// TIA Portal V17 export
// export: Created 2022-03-12T16:05:15.4162152Z, ExportSetting WithDefaults, DisplayName Totally Integrated Automation Portal, DisplayVersion V17, DisplayName TIA Portal Openness, DisplayVersion V17, DisplayName TIA Portal Version Control Interface, DisplayVersion V17, DisplayName STEP 7 Professional, DisplayVersion V17, DisplayName STEP 7 Safety, DisplayVersion V17, DisplayName WinCC Advanced / Unified PC, DisplayVersion V17
FUNCTION_BLOCK "UN_05_EventSummation"   // FB31625, LAD
TITLE = UN_05_EventSummation
{ S7_Optimized_Access := 'TRUE' }
AUTHOR : tech.team.motioncontrol@siemens.com
FAMILY : CPG
VERSION : 1.1
// Support: tech.team.motioncontrol@siemens.com
// stored: AutoNumber true, IsIECCheckEnabled false, IsRetainMemResEnabled false, MemoryReserve 100, SetENOAutomatically false, UDAEnableTagReadback false
   VAR
      instEventSumBeg_Alarm { S7_SetPoint := 'True'} : "CPG_EventSummationBegin";   // instanceFB - EventSummationBegin - Alarm Events
      instEventSum_Alarm_UN { S7_SetPoint := 'True'} : "CPG_EventSummation";   // instanceFB - EventSummation FB - Alarm Events - UN
      instEventSum_Alarm_EM00 { S7_SetPoint := 'True'} : "CPG_EventSummation";   // instanceFB - EventSummation FB - Alarm Events - EM00
      instEventSum_Alarm_EM01 { S7_SetPoint := 'True'} : "CPG_EventSummation";   // instanceFB - EventSummation FB - Alarm Events - EM01
      instEventSum_Alarm_EM02 { S7_SetPoint := 'True'} : "CPG_EventSummation";   // instanceFB - EventSummation FB - Alarm Events - EM02
      instEventSumEnd_Alarm { S7_SetPoint := 'True'} : "CPG_EventSummationEnd";   // instanceFB - EventSummationEnd - Alarm Events
      instEventSortFilter_Alarm { S7_SetPoint := 'True'} : "CPG_EventSortFilter";   // instanceFB - EventSortFilter FB - Alarms
      instAlarmMove { S7_SetPoint := 'True'} : "CPG_AlarmMove";   // instance FB - Alarm Move
      instEventSumBeg_Warning { S7_SetPoint := 'True'} : "CPG_EventSummationBegin";   // instanceFB - EventSummationBegin - Warning Events
      instEventSum_Warning_UN { S7_SetPoint := 'True'} : "CPG_EventSummation";   // instanceFB - EventSummation FB - Warning Events - UN
      instEventSum_Warning_EM00 { S7_SetPoint := 'True'} : "CPG_EventSummation";   // instanceFB - EventSummation FB - Warning Events - EM00
      instEventSum_Warning_EM01 { S7_SetPoint := 'True'} : "CPG_EventSummation";   // instanceFB - EventSummation FB - Warning Events - EM01
      instEventSum_Warning_EM02 { S7_SetPoint := 'True'} : "CPG_EventSummation";   // instanceFB - EventSummation FB - Warning Events - EM02
      instEventSumEnd_Warning { S7_SetPoint := 'True'} : "CPG_EventSummationEnd";   // instanceFB - EventSummationEnd - Warning Events
      instEventSortFilter_Warning { S7_SetPoint := 'True'} : "CPG_EventSortFilter";   // instanceFB - EventSortFilter FB - Alarms
      instWarning_MsgScroll { S7_SetPoint := 'True'} : "CPG_MsgScroll";   // instance FB - Warning Scroll
      instEventSumBeg_Status { S7_SetPoint := 'True'} : "CPG_EventSummationBegin";   // instanceFB - EventSummationBegin - Status Events
      instEventSum_Status_UN { S7_SetPoint := 'True'} : "CPG_EventSummation";   // instanceFB - EventSummation FB - Status Events - UN
      instEventSum_Status_EM00 { S7_SetPoint := 'True'} : "CPG_EventSummation";   // instanceFB - EventSummation FB - Status Events - EM00
      instEventSum_Status_EM01 { S7_SetPoint := 'True'} : "CPG_EventSummation";   // instanceFB - EventSummation FB - Status Events - EM01
      instEventSum_Status_EM02 { S7_SetPoint := 'True'} : "CPG_EventSummation";   // instanceFB - EventSummation FB - Status Events - EM02
      instEventSumEnd_Status { S7_SetPoint := 'True'} : "CPG_EventSummationEnd";   // instanceFB - EventSummationEnd - Status Events
      instPackML_AlarmHistory { S7_SetPoint := 'True'} : "CPG_AlarmHistory";   // instance FB - Capturing the 1st fault history
      instProgram_Alarm { S7_SetPoint := 'True'} : Program_Alarm;   // instance DB for Program Alarm - diag to PLC HMI
      instWarningMove { S7_SetPoint := 'True'} : "CPG_AlarmMove";
      instPareto { S7_SetPoint := 'True'} : "CPG_ParetoAnalysis";
   END_VAR
   VAR_TEMP
      tempAlarmMove_Sts_Error : Bool;   // Error with AlarmMove?
      tempAlarmMove_Sts_ErrorCode : Int;   // AlarmMove Error code
      tempProgramAlarm_error : Bool;
      tempProgramAlarm_status : Word;
   END_VAR
BEGIN

REGION Network 1: Call the Alarm Event Summary - Beginning FB
   // **********  ALARM CONTROL SUMMATION  **********
   //  
   // The event summation begin instruction prepares the summation blocks.  It should 
   // be run each time before the FB_EventSummation blocks.
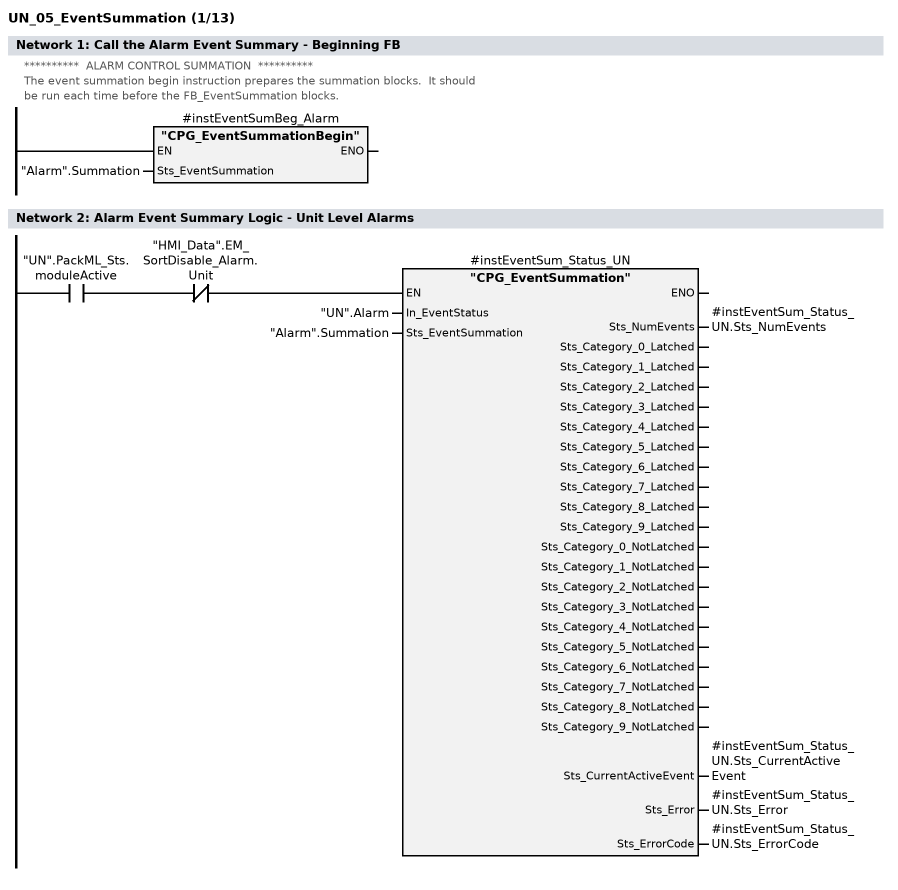
   RUNG wire#powerrail
      #instEventSumBeg_Alarm(Sts_EventSummation := "Alarm".Summation)
   END_RUNG
   // the same network as SCL:
   #instEventSumBeg_Alarm(Sts_EventSummation := "Alarm".Summation);   // "CPG_EventSummationBegin"
END_REGION

REGION Network 2: Alarm Event Summary Logic - Unit Level Alarms
   RUNG wire#powerrail
      Contact( "UN".PackML_Sts.moduleActive )
      I_Contact( "HMI_Data".EM_SortDisable_Alarm.Unit )
      #instEventSum_Status_UN(In_EventStatus := "UN".Alarm, Sts_EventSummation := "Alarm".Summation, Sts_NumEvents => #instEventSum_Status_UN.Sts_NumEvents, Sts_Category_0_Latched =>, Sts_Category_1_Latched =>, Sts_Category_2_Latched =>, Sts_Category_3_Latched =>, Sts_Category_4_Latched =>, Sts_Category_5_Latched =>, Sts_Category_6_Latched =>, Sts_Category_7_Latched =>, Sts_Category_8_Latched =>, Sts_Category_9_Latched =>, Sts_Category_0_NotLatched =>, Sts_Category_1_NotLatched =>, Sts_Category_2_NotLatched =>, Sts_Category_3_NotLatched =>, Sts_Category_4_NotLatched =>, Sts_Category_5_NotLatched =>, Sts_Category_6_NotLatched =>, Sts_Category_7_NotLatched =>, Sts_Category_8_NotLatched =>, Sts_Category_9_NotLatched =>, Sts_CurrentActiveEvent => #instEventSum_Status_UN.Sts_CurrentActiveEvent, Sts_Error => #instEventSum_Status_UN.Sts_Error, Sts_ErrorCode => #instEventSum_Status_UN.Sts_ErrorCode)
   END_RUNG
   // the same network as SCL:
   IF "UN".PackML_Sts.moduleActive AND NOT "HMI_Data".EM_SortDisable_Alarm.Unit THEN
       #instEventSum_Status_UN(In_EventStatus := "UN".Alarm,   // "CPG_EventSummation"
                               Sts_EventSummation := "Alarm".Summation,
                               Sts_NumEvents => #instEventSum_Status_UN.Sts_NumEvents,
                               Sts_CurrentActiveEvent => #instEventSum_Status_UN.Sts_CurrentActiveEvent,
                               Sts_Error => #instEventSum_Status_UN.Sts_Error,
                               Sts_ErrorCode => #instEventSum_Status_UN.Sts_ErrorCode);
   END_IF;
END_REGION

REGION Network 3: Alarm Event Summary Logic - Equipment Module #00
   // This instance of the Event Sum (or Event Summation) is used to merge the events 
   // from EM0 into the larger Unit or UN evevts list.
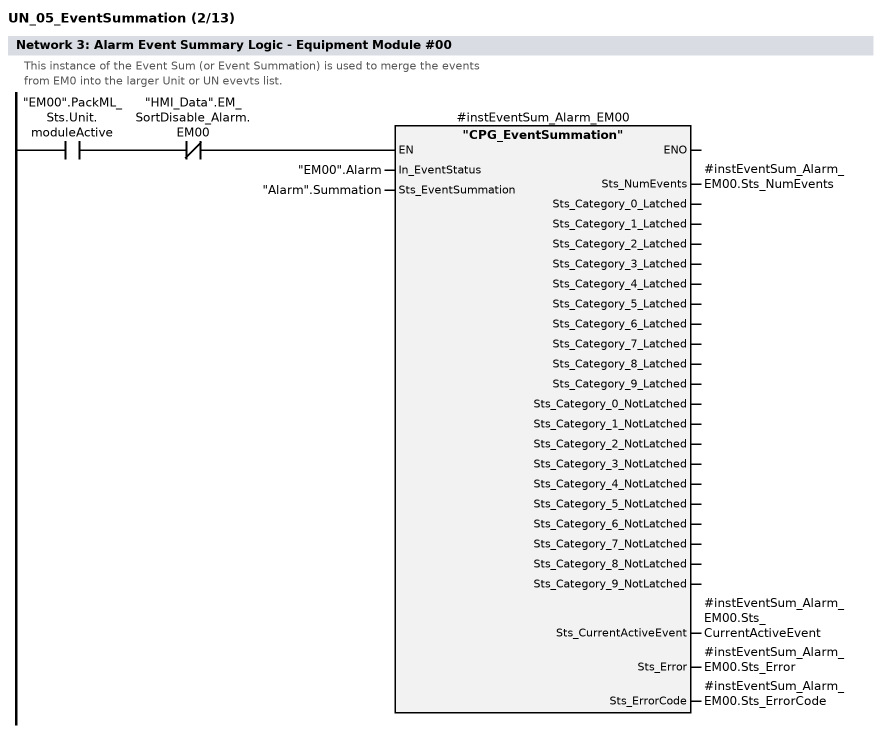
   RUNG wire#powerrail
      Contact( "EM00".PackML_Sts.Unit.moduleActive )
      I_Contact( "HMI_Data".EM_SortDisable_Alarm.EM00 )
      #instEventSum_Alarm_EM00(In_EventStatus := "EM00".Alarm, Sts_EventSummation := "Alarm".Summation, Sts_NumEvents => #instEventSum_Alarm_EM00.Sts_NumEvents, Sts_Category_0_Latched =>, Sts_Category_1_Latched =>, Sts_Category_2_Latched =>, Sts_Category_3_Latched =>, Sts_Category_4_Latched =>, Sts_Category_5_Latched =>, Sts_Category_6_Latched =>, Sts_Category_7_Latched =>, Sts_Category_8_Latched =>, Sts_Category_9_Latched =>, Sts_Category_0_NotLatched =>, Sts_Category_1_NotLatched =>, Sts_Category_2_NotLatched =>, Sts_Category_3_NotLatched =>, Sts_Category_4_NotLatched =>, Sts_Category_5_NotLatched =>, Sts_Category_6_NotLatched =>, Sts_Category_7_NotLatched =>, Sts_Category_8_NotLatched =>, Sts_Category_9_NotLatched =>, Sts_CurrentActiveEvent => #instEventSum_Alarm_EM00.Sts_CurrentActiveEvent, Sts_Error => #instEventSum_Alarm_EM00.Sts_Error, Sts_ErrorCode => #instEventSum_Alarm_EM00.Sts_ErrorCode)
   END_RUNG
   // the same network as SCL:
   IF "EM00".PackML_Sts.Unit.moduleActive AND NOT "HMI_Data".EM_SortDisable_Alarm.EM00 THEN
       #instEventSum_Alarm_EM00(In_EventStatus := "EM00".Alarm,   // "CPG_EventSummation"
                               Sts_EventSummation := "Alarm".Summation,
                               Sts_NumEvents => #instEventSum_Alarm_EM00.Sts_NumEvents,
                               Sts_CurrentActiveEvent => #instEventSum_Alarm_EM00.Sts_CurrentActiveEvent,
                               Sts_Error => #instEventSum_Alarm_EM00.Sts_Error,
                               Sts_ErrorCode => #instEventSum_Alarm_EM00.Sts_ErrorCode);
   END_IF;
END_REGION

REGION Network 4: Alarm Event Summary Logic - Equipment Module #01
   // This instance of the Event Sum (or Event Summation) is used to merge the events 
   // from EM01 into the larger Unit or UN evevts list.
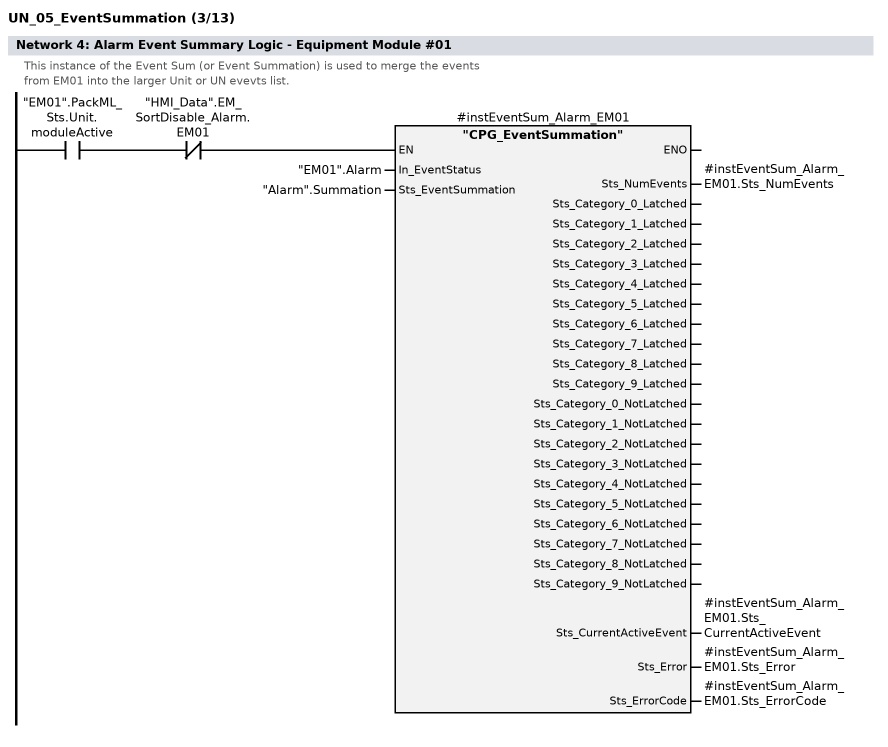
   RUNG wire#powerrail
      Contact( "EM01".PackML_Sts.Unit.moduleActive )
      I_Contact( "HMI_Data".EM_SortDisable_Alarm.EM01 )
      #instEventSum_Alarm_EM01(In_EventStatus := "EM01".Alarm, Sts_EventSummation := "Alarm".Summation, Sts_NumEvents => #instEventSum_Alarm_EM01.Sts_NumEvents, Sts_Category_0_Latched =>, Sts_Category_1_Latched =>, Sts_Category_2_Latched =>, Sts_Category_3_Latched =>, Sts_Category_4_Latched =>, Sts_Category_5_Latched =>, Sts_Category_6_Latched =>, Sts_Category_7_Latched =>, Sts_Category_8_Latched =>, Sts_Category_9_Latched =>, Sts_Category_0_NotLatched =>, Sts_Category_1_NotLatched =>, Sts_Category_2_NotLatched =>, Sts_Category_3_NotLatched =>, Sts_Category_4_NotLatched =>, Sts_Category_5_NotLatched =>, Sts_Category_6_NotLatched =>, Sts_Category_7_NotLatched =>, Sts_Category_8_NotLatched =>, Sts_Category_9_NotLatched =>, Sts_CurrentActiveEvent => #instEventSum_Alarm_EM01.Sts_CurrentActiveEvent, Sts_Error => #instEventSum_Alarm_EM01.Sts_Error, Sts_ErrorCode => #instEventSum_Alarm_EM01.Sts_ErrorCode)
   END_RUNG
   // the same network as SCL:
   IF "EM01".PackML_Sts.Unit.moduleActive AND NOT "HMI_Data".EM_SortDisable_Alarm.EM01 THEN
       #instEventSum_Alarm_EM01(In_EventStatus := "EM01".Alarm,   // "CPG_EventSummation"
                               Sts_EventSummation := "Alarm".Summation,
                               Sts_NumEvents => #instEventSum_Alarm_EM01.Sts_NumEvents,
                               Sts_CurrentActiveEvent => #instEventSum_Alarm_EM01.Sts_CurrentActiveEvent,
                               Sts_Error => #instEventSum_Alarm_EM01.Sts_Error,
                               Sts_ErrorCode => #instEventSum_Alarm_EM01.Sts_ErrorCode);
   END_IF;
END_REGION

REGION Network 5: Alarm Event Summary Logic - Equipment Module #02
   // This instance of the Event Sum (or Event Summation) is used to merge the events 
   // from EM01 into the larger Unit or UN evevts list.
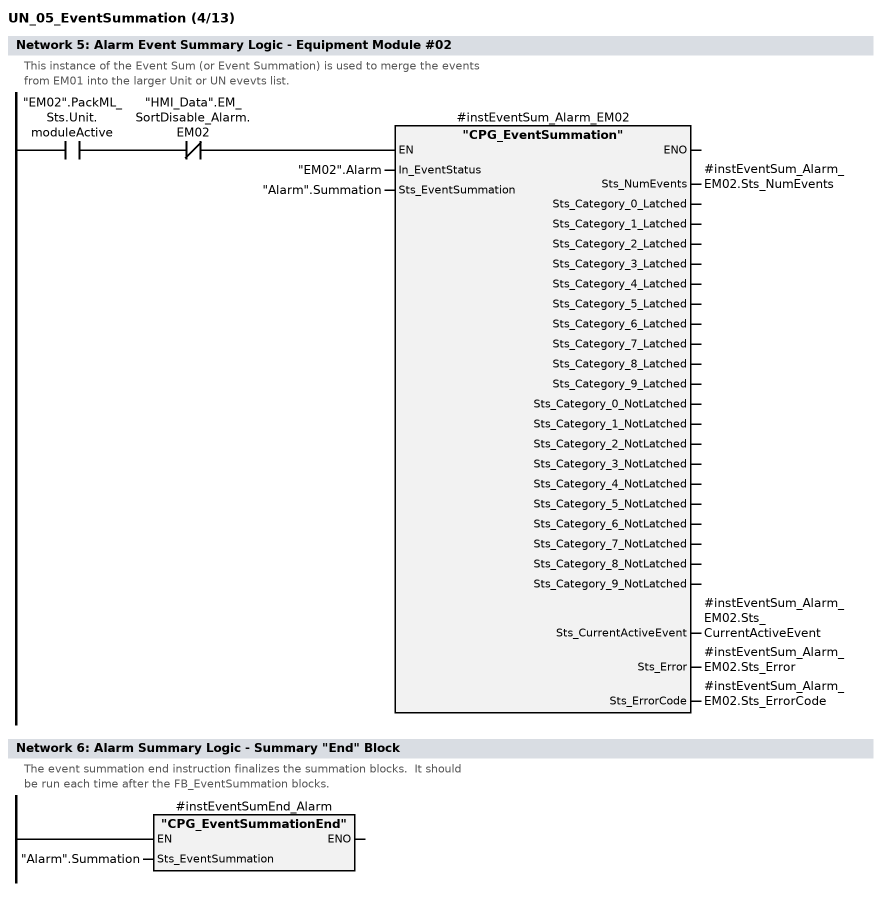
   RUNG wire#powerrail
      Contact( "EM02".PackML_Sts.Unit.moduleActive )
      I_Contact( "HMI_Data".EM_SortDisable_Alarm.EM02 )
      #instEventSum_Alarm_EM02(In_EventStatus := "EM02".Alarm, Sts_EventSummation := "Alarm".Summation, Sts_NumEvents => #instEventSum_Alarm_EM02.Sts_NumEvents, Sts_Category_0_Latched =>, Sts_Category_1_Latched =>, Sts_Category_2_Latched =>, Sts_Category_3_Latched =>, Sts_Category_4_Latched =>, Sts_Category_5_Latched =>, Sts_Category_6_Latched =>, Sts_Category_7_Latched =>, Sts_Category_8_Latched =>, Sts_Category_9_Latched =>, Sts_Category_0_NotLatched =>, Sts_Category_1_NotLatched =>, Sts_Category_2_NotLatched =>, Sts_Category_3_NotLatched =>, Sts_Category_4_NotLatched =>, Sts_Category_5_NotLatched =>, Sts_Category_6_NotLatched =>, Sts_Category_7_NotLatched =>, Sts_Category_8_NotLatched =>, Sts_Category_9_NotLatched =>, Sts_CurrentActiveEvent => #instEventSum_Alarm_EM02.Sts_CurrentActiveEvent, Sts_Error => #instEventSum_Alarm_EM02.Sts_Error, Sts_ErrorCode => #instEventSum_Alarm_EM02.Sts_ErrorCode)
   END_RUNG
   // the same network as SCL:
   IF "EM02".PackML_Sts.Unit.moduleActive AND NOT "HMI_Data".EM_SortDisable_Alarm.EM02 THEN
       #instEventSum_Alarm_EM02(In_EventStatus := "EM02".Alarm,   // "CPG_EventSummation"
                               Sts_EventSummation := "Alarm".Summation,
                               Sts_NumEvents => #instEventSum_Alarm_EM02.Sts_NumEvents,
                               Sts_CurrentActiveEvent => #instEventSum_Alarm_EM02.Sts_CurrentActiveEvent,
                               Sts_Error => #instEventSum_Alarm_EM02.Sts_Error,
                               Sts_ErrorCode => #instEventSum_Alarm_EM02.Sts_ErrorCode);
   END_IF;
END_REGION

REGION Network 6: Alarm Summary Logic - Summary "End" Block
   // The event summation end instruction finalizes the summation blocks.  It should 
   // be run each time after the FB_EventSummation blocks.
   RUNG wire#powerrail
      #instEventSumEnd_Alarm(Sts_EventSummation := "Alarm".Summation)
   END_RUNG
   // the same network as SCL:
   #instEventSumEnd_Alarm(Sts_EventSummation := "Alarm".Summation);   // "CPG_EventSummationEnd"
END_REGION

REGION Network 7: Update Admin.Alarm information.
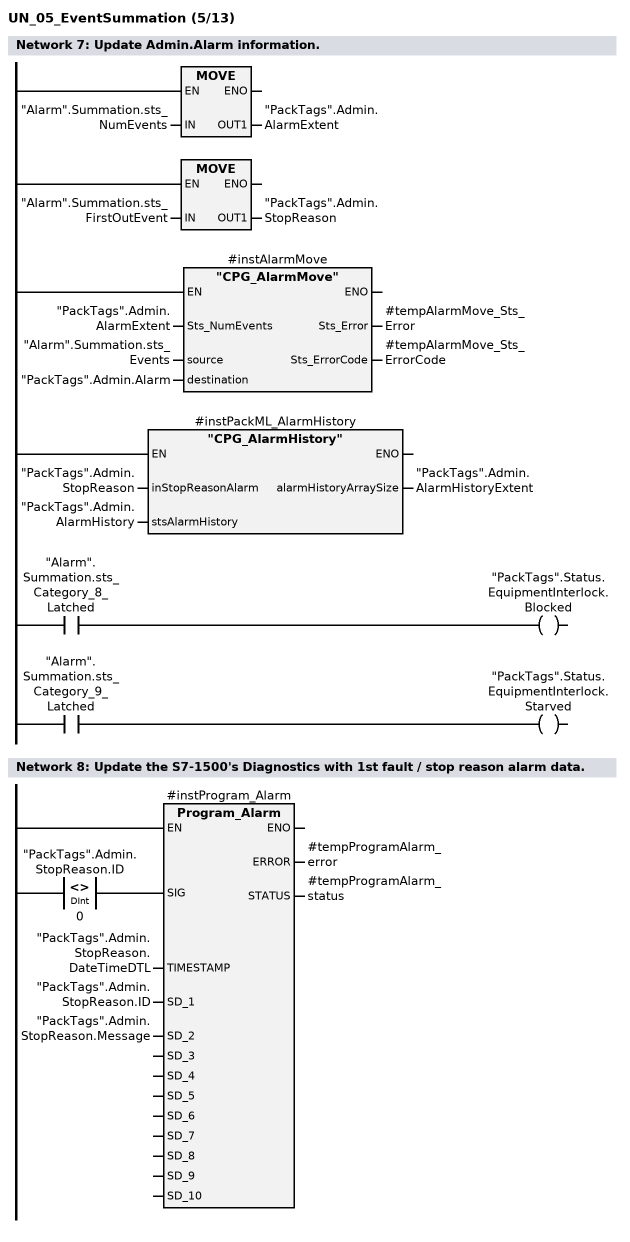
   RUNG wire#powerrail
      { S7_GenerateENO := "TRUE" } Move(in := "Alarm".Summation.sts_NumEvents, out1 => "PackTags".Admin.AlarmExtent)
   END_RUNG
   RUNG wire#powerrail
      Move(in := "Alarm".Summation.sts_FirstOutEvent, out1 => "PackTags".Admin.StopReason)
   END_RUNG
   RUNG wire#powerrail
      #instAlarmMove(Sts_NumEvents := "PackTags".Admin.AlarmExtent, source := "Alarm".Summation.sts_Events, destination := "PackTags".Admin.Alarm, Sts_Error => #tempAlarmMove_Sts_Error, Sts_ErrorCode => #tempAlarmMove_Sts_ErrorCode)
   END_RUNG
   RUNG wire#powerrail
      #instPackML_AlarmHistory(inStopReasonAlarm := "PackTags".Admin.StopReason, stsAlarmHistory := "PackTags".Admin.AlarmHistory, alarmHistoryArraySize => "PackTags".Admin.AlarmHistoryExtent)
   END_RUNG
   RUNG wire#powerrail
      Contact( "Alarm".Summation.sts_Category_8_Latched )
      Coil( "PackTags".Status.EquipmentInterlock.Blocked )
   END_RUNG
   RUNG wire#powerrail
      Contact( "Alarm".Summation.sts_Category_9_Latched )
      Coil( "PackTags".Status.EquipmentInterlock.Starved )
   END_RUNG
   // the same network as SCL:
   "PackTags".Admin.AlarmExtent := "Alarm".Summation.sts_NumEvents;
   "PackTags".Admin.StopReason := "Alarm".Summation.sts_FirstOutEvent;
   #instAlarmMove(Sts_NumEvents := "PackTags".Admin.AlarmExtent,   // "CPG_AlarmMove"
                  source := "Alarm".Summation.sts_Events,
                  destination := "PackTags".Admin.Alarm,
                  Sts_Error => #tempAlarmMove_Sts_Error,
                  Sts_ErrorCode => #tempAlarmMove_Sts_ErrorCode);
   #instPackML_AlarmHistory(inStopReasonAlarm := "PackTags".Admin.StopReason,   // "CPG_AlarmHistory"
                           stsAlarmHistory := "PackTags".Admin.AlarmHistory,
                           alarmHistoryArraySize => "PackTags".Admin.AlarmHistoryExtent);
   "PackTags".Status.EquipmentInterlock.Blocked := "Alarm".Summation.sts_Category_8_Latched;
   "PackTags".Status.EquipmentInterlock.Starved := "Alarm".Summation.sts_Category_9_Latched;
END_REGION

REGION Network 8: Update the S7-1500's Diagnostics with 1st fault / stop reason alarm data.
   RUNG wire#powerrail
      #instProgram_Alarm.Program_Alarm(SIG := wire#w1, TIMESTAMP := "PackTags".Admin.StopReason.DateTimeDTL, SD_1 := "PackTags".Admin.StopReason.ID, SD_2 := "PackTags".Admin.StopReason.Message, SD_3 :=, SD_4 :=, SD_5 :=, SD_6 :=, SD_7 :=, SD_8 :=, SD_9 :=, SD_10 :=, Error => #tempProgramAlarm_error, Status => #tempProgramAlarm_status)
   END_RUNG
   RUNG wire#powerrail
      { S7_Templates := "SrcType := DInt" } NE_Contact(in1 := "PackTags".Admin.StopReason.ID, in2 := 0)
   END_RUNG wire#w1
   // the same network as SCL:
   #instProgram_Alarm(SIG := "PackTags".Admin.StopReason.ID <> 0,   // Program_Alarm
                      TIMESTAMP := "PackTags".Admin.StopReason.DateTimeDTL,
                      SD_1 := "PackTags".Admin.StopReason.ID,
                      SD_2 := "PackTags".Admin.StopReason.Message,
                      Error => #tempProgramAlarm_error,
                      Status => #tempProgramAlarm_status);
END_REGION

REGION Network 9: Event Sort Filter logic - Alarms
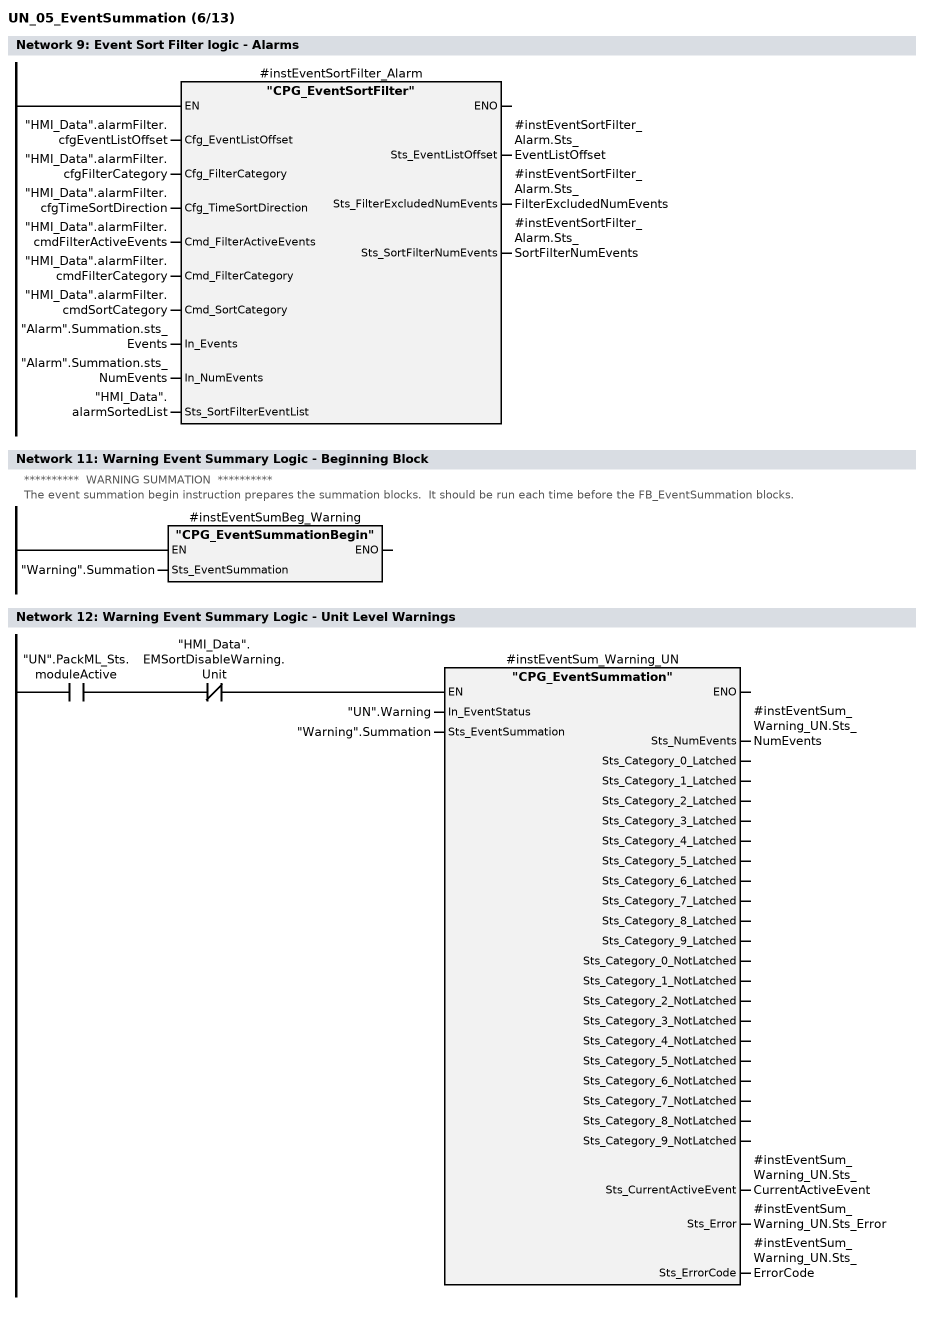
   RUNG wire#powerrail
      #instEventSortFilter_Alarm(Cfg_EventListOffset := "HMI_Data".alarmFilter.cfgEventListOffset, Cfg_FilterCategory := "HMI_Data".alarmFilter.cfgFilterCategory, Cfg_TimeSortDirection := "HMI_Data".alarmFilter.cfgTimeSortDirection, Cmd_FilterActiveEvents := "HMI_Data".alarmFilter.cmdFilterActiveEvents, Cmd_FilterCategory := "HMI_Data".alarmFilter.cmdFilterCategory, Cmd_SortCategory := "HMI_Data".alarmFilter.cmdSortCategory, In_Events := "Alarm".Summation.sts_Events, In_NumEvents := "Alarm".Summation.sts_NumEvents, Sts_SortFilterEventList := "HMI_Data".alarmSortedList, Sts_EventListOffset => #instEventSortFilter_Alarm.Sts_EventListOffset, Sts_FilterExcludedNumEvents => #instEventSortFilter_Alarm.Sts_FilterExcludedNumEvents, Sts_SortFilterNumEvents => #instEventSortFilter_Alarm.Sts_SortFilterNumEvents)
   END_RUNG
   // the same network as SCL:
   #instEventSortFilter_Alarm(Cfg_EventListOffset := "HMI_Data".alarmFilter.cfgEventListOffset,   // "CPG_EventSortFilter"
                           Cfg_FilterCategory := "HMI_Data".alarmFilter.cfgFilterCategory,
                           Cfg_TimeSortDirection := "HMI_Data".alarmFilter.cfgTimeSortDirection,
                           Cmd_FilterActiveEvents := "HMI_Data".alarmFilter.cmdFilterActiveEvents,
                           Cmd_FilterCategory := "HMI_Data".alarmFilter.cmdFilterCategory,
                           Cmd_SortCategory := "HMI_Data".alarmFilter.cmdSortCategory,
                           In_Events := "Alarm".Summation.sts_Events,
                           In_NumEvents := "Alarm".Summation.sts_NumEvents,
                           Sts_SortFilterEventList := "HMI_Data".alarmSortedList,
                           Sts_EventListOffset => #instEventSortFilter_Alarm.Sts_EventListOffset,
                           Sts_FilterExcludedNumEvents => #instEventSortFilter_Alarm.Sts_FilterExcludedNumEvents,
                           Sts_SortFilterNumEvents => #instEventSortFilter_Alarm.Sts_SortFilterNumEvents);
END_REGION

REGION Network 10: *** Beging the WARNING area ****
END_REGION

REGION Network 11: Warning Event Summary Logic - Beginning Block
   // **********  WARNING SUMMATION  **********
   //  
   // The event summation begin instruction prepares the summation blocks.  It should be run each time before the FB_EventSummation blocks.
   RUNG wire#powerrail
      #instEventSumBeg_Warning(Sts_EventSummation := "Warning".Summation)
   END_RUNG
   // the same network as SCL:
   #instEventSumBeg_Warning(Sts_EventSummation := "Warning".Summation);   // "CPG_EventSummationBegin"
END_REGION

REGION Network 12: Warning Event Summary Logic - Unit Level Warnings
   RUNG wire#powerrail
      Contact( "UN".PackML_Sts.moduleActive )
      I_Contact( "HMI_Data".EMSortDisableWarning.Unit )
      #instEventSum_Warning_UN(In_EventStatus := "UN".Warning, Sts_EventSummation := "Warning".Summation, Sts_NumEvents => #instEventSum_Warning_UN.Sts_NumEvents, Sts_Category_0_Latched =>, Sts_Category_1_Latched =>, Sts_Category_2_Latched =>, Sts_Category_3_Latched =>, Sts_Category_4_Latched =>, Sts_Category_5_Latched =>, Sts_Category_6_Latched =>, Sts_Category_7_Latched =>, Sts_Category_8_Latched =>, Sts_Category_9_Latched =>, Sts_Category_0_NotLatched =>, Sts_Category_1_NotLatched =>, Sts_Category_2_NotLatched =>, Sts_Category_3_NotLatched =>, Sts_Category_4_NotLatched =>, Sts_Category_5_NotLatched =>, Sts_Category_6_NotLatched =>, Sts_Category_7_NotLatched =>, Sts_Category_8_NotLatched =>, Sts_Category_9_NotLatched =>, Sts_CurrentActiveEvent => #instEventSum_Warning_UN.Sts_CurrentActiveEvent, Sts_Error => #instEventSum_Warning_UN.Sts_Error, Sts_ErrorCode => #instEventSum_Warning_UN.Sts_ErrorCode)
   END_RUNG
   // the same network as SCL:
   IF "UN".PackML_Sts.moduleActive AND NOT "HMI_Data".EMSortDisableWarning.Unit THEN
       #instEventSum_Warning_UN(In_EventStatus := "UN".Warning,   // "CPG_EventSummation"
                               Sts_EventSummation := "Warning".Summation,
                               Sts_NumEvents => #instEventSum_Warning_UN.Sts_NumEvents,
                               Sts_CurrentActiveEvent => #instEventSum_Warning_UN.Sts_CurrentActiveEvent,
                               Sts_Error => #instEventSum_Warning_UN.Sts_Error,
                               Sts_ErrorCode => #instEventSum_Warning_UN.Sts_ErrorCode);
   END_IF;
END_REGION

REGION Network 13: Warning Event Summary Logic - Equipment Module #00
   // This instance of the Event Sum (or Event Summation) is used to merge the events 
   // from EM0 into the larger Unit or UN evevts list.
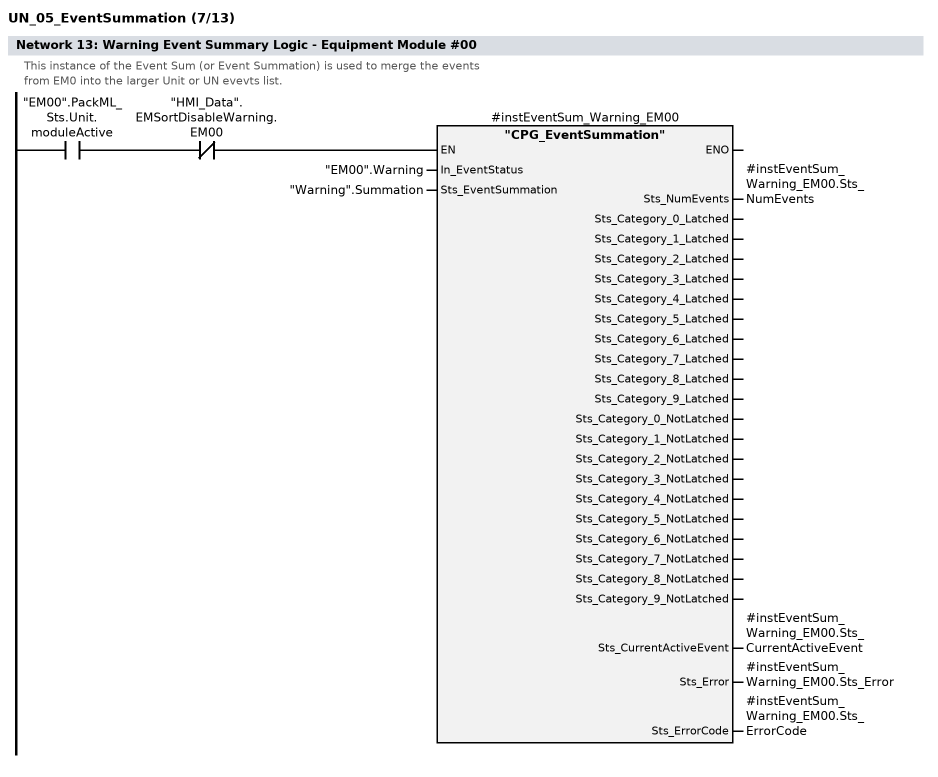
   RUNG wire#powerrail
      Contact( "EM00".PackML_Sts.Unit.moduleActive )
      I_Contact( "HMI_Data".EMSortDisableWarning.EM00 )
      #instEventSum_Warning_EM00(In_EventStatus := "EM00".Warning, Sts_EventSummation := "Warning".Summation, Sts_NumEvents => #instEventSum_Warning_EM00.Sts_NumEvents, Sts_Category_0_Latched =>, Sts_Category_1_Latched =>, Sts_Category_2_Latched =>, Sts_Category_3_Latched =>, Sts_Category_4_Latched =>, Sts_Category_5_Latched =>, Sts_Category_6_Latched =>, Sts_Category_7_Latched =>, Sts_Category_8_Latched =>, Sts_Category_9_Latched =>, Sts_Category_0_NotLatched =>, Sts_Category_1_NotLatched =>, Sts_Category_2_NotLatched =>, Sts_Category_3_NotLatched =>, Sts_Category_4_NotLatched =>, Sts_Category_5_NotLatched =>, Sts_Category_6_NotLatched =>, Sts_Category_7_NotLatched =>, Sts_Category_8_NotLatched =>, Sts_Category_9_NotLatched =>, Sts_CurrentActiveEvent => #instEventSum_Warning_EM00.Sts_CurrentActiveEvent, Sts_Error => #instEventSum_Warning_EM00.Sts_Error, Sts_ErrorCode => #instEventSum_Warning_EM00.Sts_ErrorCode)
   END_RUNG
   // the same network as SCL:
   IF "EM00".PackML_Sts.Unit.moduleActive AND NOT "HMI_Data".EMSortDisableWarning.EM00 THEN
       #instEventSum_Warning_EM00(In_EventStatus := "EM00".Warning,   // "CPG_EventSummation"
                               Sts_EventSummation := "Warning".Summation,
                               Sts_NumEvents => #instEventSum_Warning_EM00.Sts_NumEvents,
                               Sts_CurrentActiveEvent => #instEventSum_Warning_EM00.Sts_CurrentActiveEvent,
                               Sts_Error => #instEventSum_Warning_EM00.Sts_Error,
                               Sts_ErrorCode => #instEventSum_Warning_EM00.Sts_ErrorCode);
   END_IF;
END_REGION

REGION Network 14: Warning Event Summary Logic - Equipment Module #01
   // This instance of the Event Sum (or Event Summation) is used to merge the events 
   // from EM1 into the larger Unit or UN evevts list.
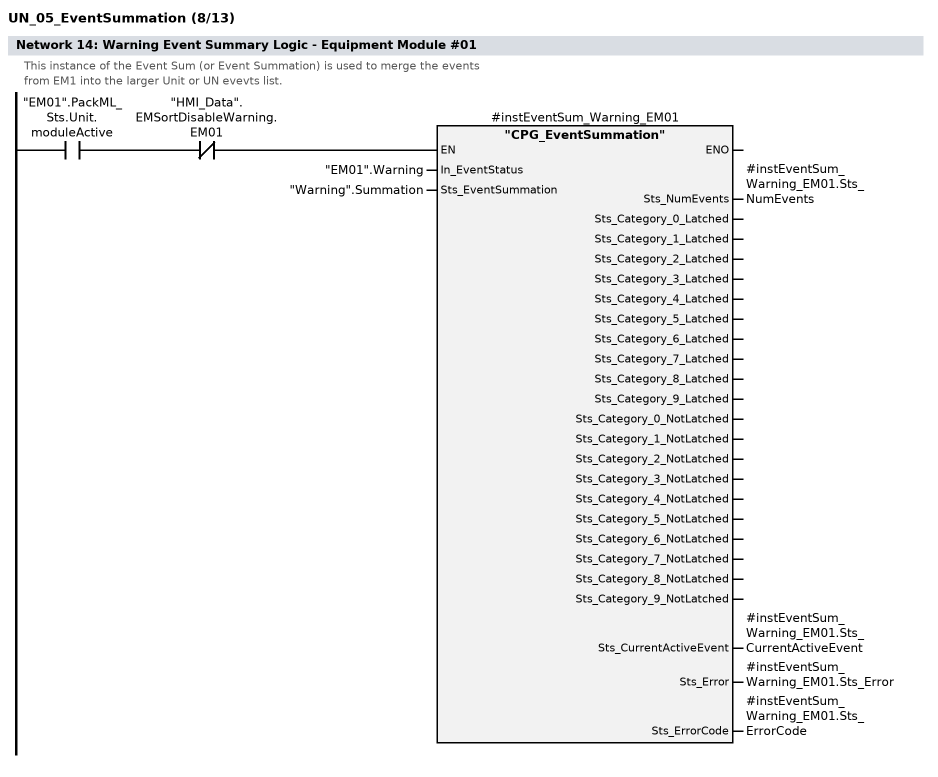
   RUNG wire#powerrail
      Contact( "EM01".PackML_Sts.Unit.moduleActive )
      I_Contact( "HMI_Data".EMSortDisableWarning.EM01 )
      #instEventSum_Warning_EM01(In_EventStatus := "EM01".Warning, Sts_EventSummation := "Warning".Summation, Sts_NumEvents => #instEventSum_Warning_EM01.Sts_NumEvents, Sts_Category_0_Latched =>, Sts_Category_1_Latched =>, Sts_Category_2_Latched =>, Sts_Category_3_Latched =>, Sts_Category_4_Latched =>, Sts_Category_5_Latched =>, Sts_Category_6_Latched =>, Sts_Category_7_Latched =>, Sts_Category_8_Latched =>, Sts_Category_9_Latched =>, Sts_Category_0_NotLatched =>, Sts_Category_1_NotLatched =>, Sts_Category_2_NotLatched =>, Sts_Category_3_NotLatched =>, Sts_Category_4_NotLatched =>, Sts_Category_5_NotLatched =>, Sts_Category_6_NotLatched =>, Sts_Category_7_NotLatched =>, Sts_Category_8_NotLatched =>, Sts_Category_9_NotLatched =>, Sts_CurrentActiveEvent => #instEventSum_Warning_EM01.Sts_CurrentActiveEvent, Sts_Error => #instEventSum_Warning_EM01.Sts_Error, Sts_ErrorCode => #instEventSum_Warning_EM01.Sts_ErrorCode)
   END_RUNG
   // the same network as SCL:
   IF "EM01".PackML_Sts.Unit.moduleActive AND NOT "HMI_Data".EMSortDisableWarning.EM01 THEN
       #instEventSum_Warning_EM01(In_EventStatus := "EM01".Warning,   // "CPG_EventSummation"
                               Sts_EventSummation := "Warning".Summation,
                               Sts_NumEvents => #instEventSum_Warning_EM01.Sts_NumEvents,
                               Sts_CurrentActiveEvent => #instEventSum_Warning_EM01.Sts_CurrentActiveEvent,
                               Sts_Error => #instEventSum_Warning_EM01.Sts_Error,
                               Sts_ErrorCode => #instEventSum_Warning_EM01.Sts_ErrorCode);
   END_IF;
END_REGION

REGION Network 15: Warning Event Summary Logic - Equipment Module #02
   // This instance of the Event Sum (or Event Summation) is used to merge the events 
   // from EM01 into the larger Unit or UN evevts list.
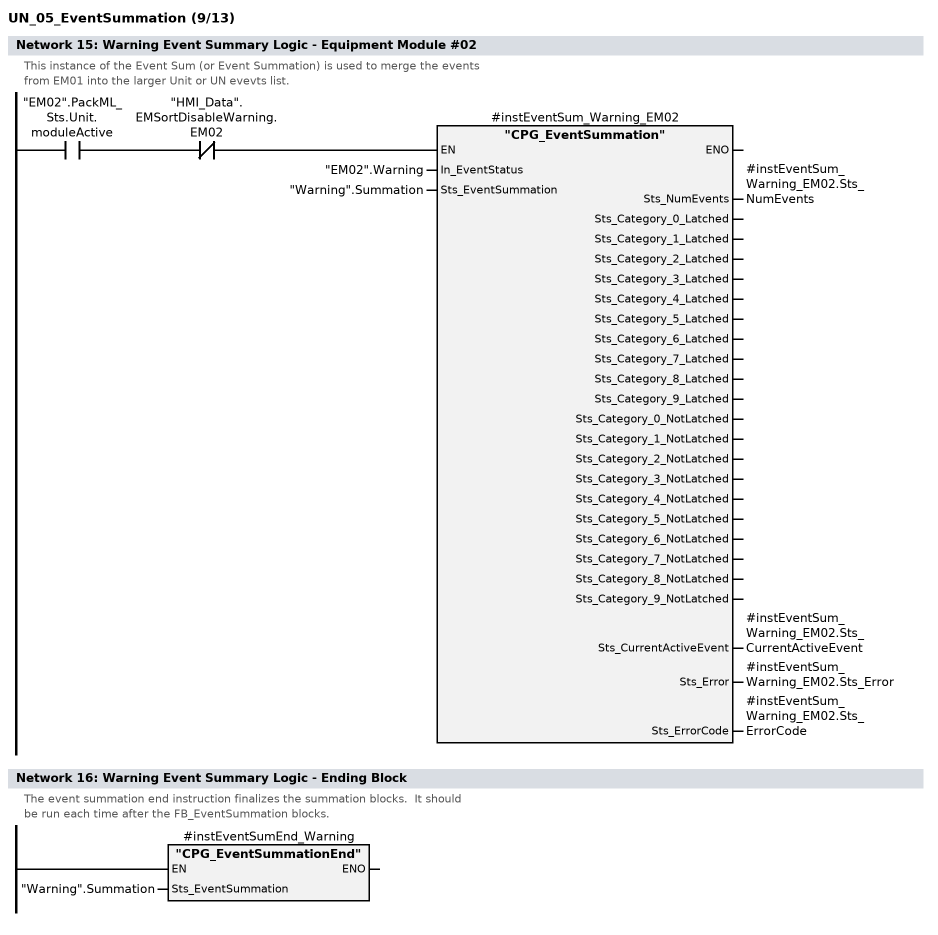
   RUNG wire#powerrail
      Contact( "EM02".PackML_Sts.Unit.moduleActive )
      I_Contact( "HMI_Data".EMSortDisableWarning.EM02 )
      #instEventSum_Warning_EM02(In_EventStatus := "EM02".Warning, Sts_EventSummation := "Warning".Summation, Sts_NumEvents => #instEventSum_Warning_EM02.Sts_NumEvents, Sts_Category_0_Latched =>, Sts_Category_1_Latched =>, Sts_Category_2_Latched =>, Sts_Category_3_Latched =>, Sts_Category_4_Latched =>, Sts_Category_5_Latched =>, Sts_Category_6_Latched =>, Sts_Category_7_Latched =>, Sts_Category_8_Latched =>, Sts_Category_9_Latched =>, Sts_Category_0_NotLatched =>, Sts_Category_1_NotLatched =>, Sts_Category_2_NotLatched =>, Sts_Category_3_NotLatched =>, Sts_Category_4_NotLatched =>, Sts_Category_5_NotLatched =>, Sts_Category_6_NotLatched =>, Sts_Category_7_NotLatched =>, Sts_Category_8_NotLatched =>, Sts_Category_9_NotLatched =>, Sts_CurrentActiveEvent => #instEventSum_Warning_EM02.Sts_CurrentActiveEvent, Sts_Error => #instEventSum_Warning_EM02.Sts_Error, Sts_ErrorCode => #instEventSum_Warning_EM02.Sts_ErrorCode)
   END_RUNG
   // the same network as SCL:
   IF "EM02".PackML_Sts.Unit.moduleActive AND NOT "HMI_Data".EMSortDisableWarning.EM02 THEN
       #instEventSum_Warning_EM02(In_EventStatus := "EM02".Warning,   // "CPG_EventSummation"
                               Sts_EventSummation := "Warning".Summation,
                               Sts_NumEvents => #instEventSum_Warning_EM02.Sts_NumEvents,
                               Sts_CurrentActiveEvent => #instEventSum_Warning_EM02.Sts_CurrentActiveEvent,
                               Sts_Error => #instEventSum_Warning_EM02.Sts_Error,
                               Sts_ErrorCode => #instEventSum_Warning_EM02.Sts_ErrorCode);
   END_IF;
END_REGION

REGION Network 16: Warning Event Summary Logic - Ending Block
   // The event summation end instruction finalizes the summation blocks.  It should 
   // be run each time after the FB_EventSummation blocks.
   RUNG wire#powerrail
      #instEventSumEnd_Warning(Sts_EventSummation := "Warning".Summation)
   END_RUNG
   // the same network as SCL:
   #instEventSumEnd_Warning(Sts_EventSummation := "Warning".Summation);   // "CPG_EventSummationEnd"
END_REGION

REGION Network 17: Event Sort Filter logic - Warnings
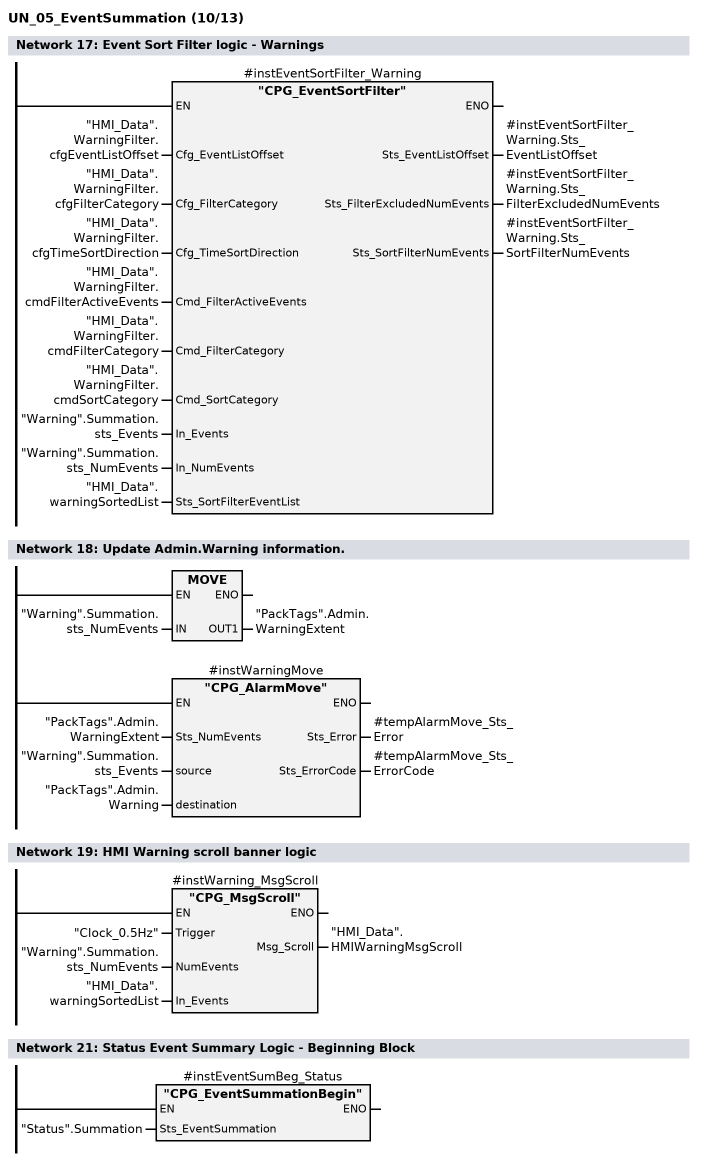
   RUNG wire#powerrail
      #instEventSortFilter_Warning(Cfg_EventListOffset := "HMI_Data".WarningFilter.cfgEventListOffset, Cfg_FilterCategory := "HMI_Data".WarningFilter.cfgFilterCategory, Cfg_TimeSortDirection := "HMI_Data".WarningFilter.cfgTimeSortDirection, Cmd_FilterActiveEvents := "HMI_Data".WarningFilter.cmdFilterActiveEvents, Cmd_FilterCategory := "HMI_Data".WarningFilter.cmdFilterCategory, Cmd_SortCategory := "HMI_Data".WarningFilter.cmdSortCategory, In_Events := "Warning".Summation.sts_Events, In_NumEvents := "Warning".Summation.sts_NumEvents, Sts_SortFilterEventList := "HMI_Data".warningSortedList, Sts_EventListOffset => #instEventSortFilter_Warning.Sts_EventListOffset, Sts_FilterExcludedNumEvents => #instEventSortFilter_Warning.Sts_FilterExcludedNumEvents, Sts_SortFilterNumEvents => #instEventSortFilter_Warning.Sts_SortFilterNumEvents)
   END_RUNG
   // the same network as SCL:
   #instEventSortFilter_Warning(Cfg_EventListOffset := "HMI_Data".WarningFilter.cfgEventListOffset,   // "CPG_EventSortFilter"
                           Cfg_FilterCategory := "HMI_Data".WarningFilter.cfgFilterCategory,
                           Cfg_TimeSortDirection := "HMI_Data".WarningFilter.cfgTimeSortDirection,
                           Cmd_FilterActiveEvents := "HMI_Data".WarningFilter.cmdFilterActiveEvents,
                           Cmd_FilterCategory := "HMI_Data".WarningFilter.cmdFilterCategory,
                           Cmd_SortCategory := "HMI_Data".WarningFilter.cmdSortCategory,
                           In_Events := "Warning".Summation.sts_Events,
                           In_NumEvents := "Warning".Summation.sts_NumEvents,
                           Sts_SortFilterEventList := "HMI_Data".warningSortedList,
                           Sts_EventListOffset => #instEventSortFilter_Warning.Sts_EventListOffset,
                           Sts_FilterExcludedNumEvents => #instEventSortFilter_Warning.Sts_FilterExcludedNumEvents,
                           Sts_SortFilterNumEvents => #instEventSortFilter_Warning.Sts_SortFilterNumEvents);
END_REGION

REGION Network 18: Update Admin.Warning information.
   RUNG wire#powerrail
      { S7_GenerateENO := "TRUE" } Move(in := "Warning".Summation.sts_NumEvents, out1 => "PackTags".Admin.WarningExtent)
   END_RUNG
   RUNG wire#powerrail
      #instWarningMove(Sts_NumEvents := "PackTags".Admin.WarningExtent, source := "Warning".Summation.sts_Events, destination := "PackTags".Admin.Warning, Sts_Error => #tempAlarmMove_Sts_Error, Sts_ErrorCode => #tempAlarmMove_Sts_ErrorCode)
   END_RUNG
   // the same network as SCL:
   "PackTags".Admin.WarningExtent := "Warning".Summation.sts_NumEvents;
   #instWarningMove(Sts_NumEvents := "PackTags".Admin.WarningExtent,   // "CPG_AlarmMove"
                    source := "Warning".Summation.sts_Events,
                    destination := "PackTags".Admin.Warning,
                    Sts_Error => #tempAlarmMove_Sts_Error,
                    Sts_ErrorCode => #tempAlarmMove_Sts_ErrorCode);
END_REGION

REGION Network 19: HMI Warning scroll banner logic
   RUNG wire#powerrail
      #instWarning_MsgScroll(Trigger := "Clock_0.5Hz", NumEvents := "Warning".Summation.sts_NumEvents, In_Events := "HMI_Data".warningSortedList, Msg_Scroll => "HMI_Data".HMIWarningMsgScroll)
   END_RUNG
   // the same network as SCL:
   #instWarning_MsgScroll(Trigger := "Clock_0.5Hz",   // "CPG_MsgScroll"
                          NumEvents := "Warning".Summation.sts_NumEvents,
                          In_Events := "HMI_Data".warningSortedList,
                          Msg_Scroll => "HMI_Data".HMIWarningMsgScroll);
END_REGION

REGION Network 20: *** Status Event Summation ***
END_REGION

REGION Network 21: Status Event Summary Logic - Beginning Block
   RUNG wire#powerrail
      #instEventSumBeg_Status(Sts_EventSummation := "Status".Summation)
   END_RUNG
   // the same network as SCL:
   #instEventSumBeg_Status(Sts_EventSummation := "Status".Summation);   // "CPG_EventSummationBegin"
END_REGION

REGION Network 22: Status Event Summary Logic - Unit
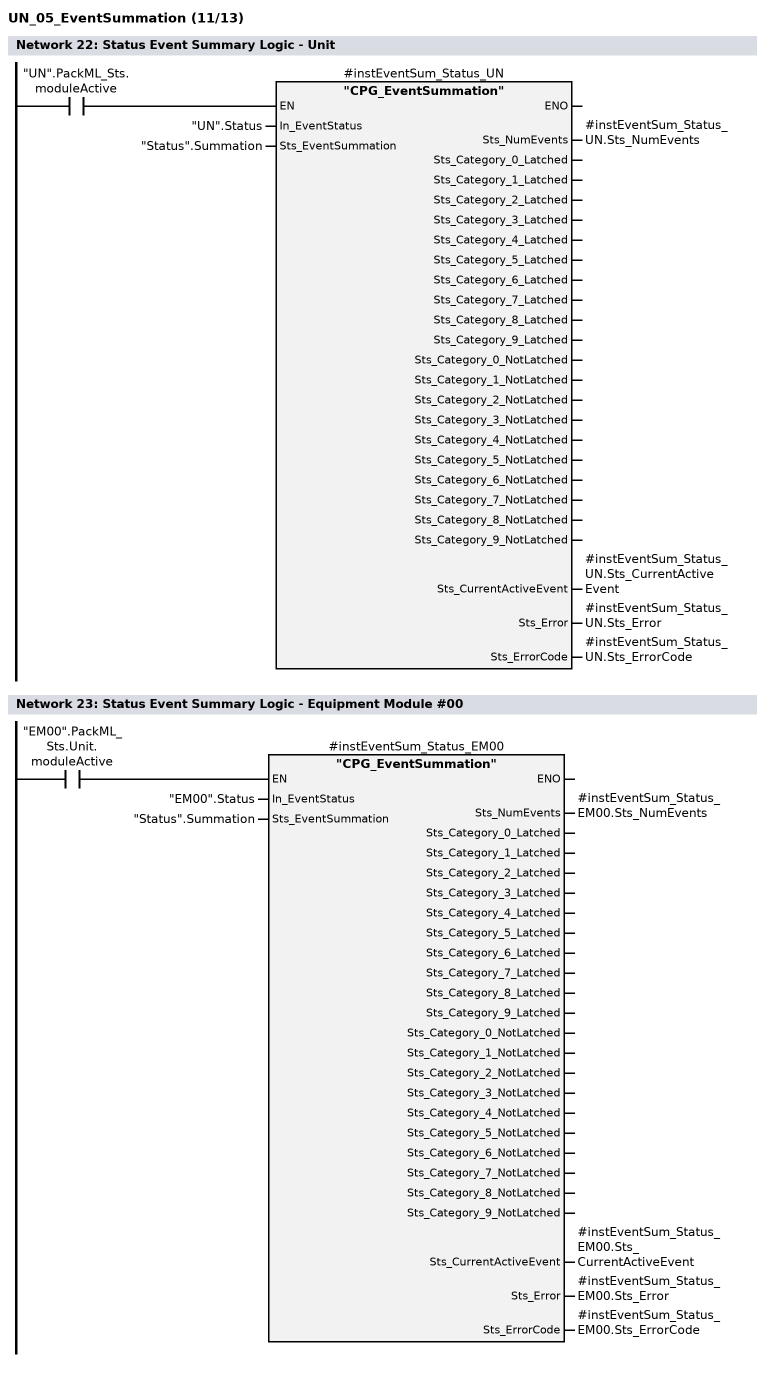
   RUNG wire#powerrail
      Contact( "UN".PackML_Sts.moduleActive )
      #instEventSum_Status_UN(In_EventStatus := "UN".Status, Sts_EventSummation := "Status".Summation, Sts_NumEvents => #instEventSum_Status_UN.Sts_NumEvents, Sts_Category_0_Latched =>, Sts_Category_1_Latched =>, Sts_Category_2_Latched =>, Sts_Category_3_Latched =>, Sts_Category_4_Latched =>, Sts_Category_5_Latched =>, Sts_Category_6_Latched =>, Sts_Category_7_Latched =>, Sts_Category_8_Latched =>, Sts_Category_9_Latched =>, Sts_Category_0_NotLatched =>, Sts_Category_1_NotLatched =>, Sts_Category_2_NotLatched =>, Sts_Category_3_NotLatched =>, Sts_Category_4_NotLatched =>, Sts_Category_5_NotLatched =>, Sts_Category_6_NotLatched =>, Sts_Category_7_NotLatched =>, Sts_Category_8_NotLatched =>, Sts_Category_9_NotLatched =>, Sts_CurrentActiveEvent => #instEventSum_Status_UN.Sts_CurrentActiveEvent, Sts_Error => #instEventSum_Status_UN.Sts_Error, Sts_ErrorCode => #instEventSum_Status_UN.Sts_ErrorCode)
   END_RUNG
   // the same network as SCL:
   IF "UN".PackML_Sts.moduleActive THEN
       #instEventSum_Status_UN(In_EventStatus := "UN".Status,   // "CPG_EventSummation"
                               Sts_EventSummation := "Status".Summation,
                               Sts_NumEvents => #instEventSum_Status_UN.Sts_NumEvents,
                               Sts_CurrentActiveEvent => #instEventSum_Status_UN.Sts_CurrentActiveEvent,
                               Sts_Error => #instEventSum_Status_UN.Sts_Error,
                               Sts_ErrorCode => #instEventSum_Status_UN.Sts_ErrorCode);
   END_IF;
END_REGION

REGION Network 23: Status Event Summary Logic - Equipment Module #00
   RUNG wire#powerrail
      Contact( "EM00".PackML_Sts.Unit.moduleActive )
      #instEventSum_Status_EM00(In_EventStatus := "EM00".Status, Sts_EventSummation := "Status".Summation, Sts_NumEvents => #instEventSum_Status_EM00.Sts_NumEvents, Sts_Category_0_Latched =>, Sts_Category_1_Latched =>, Sts_Category_2_Latched =>, Sts_Category_3_Latched =>, Sts_Category_4_Latched =>, Sts_Category_5_Latched =>, Sts_Category_6_Latched =>, Sts_Category_7_Latched =>, Sts_Category_8_Latched =>, Sts_Category_9_Latched =>, Sts_Category_0_NotLatched =>, Sts_Category_1_NotLatched =>, Sts_Category_2_NotLatched =>, Sts_Category_3_NotLatched =>, Sts_Category_4_NotLatched =>, Sts_Category_5_NotLatched =>, Sts_Category_6_NotLatched =>, Sts_Category_7_NotLatched =>, Sts_Category_8_NotLatched =>, Sts_Category_9_NotLatched =>, Sts_CurrentActiveEvent => #instEventSum_Status_EM00.Sts_CurrentActiveEvent, Sts_Error => #instEventSum_Status_EM00.Sts_Error, Sts_ErrorCode => #instEventSum_Status_EM00.Sts_ErrorCode)
   END_RUNG
   // the same network as SCL:
   IF "EM00".PackML_Sts.Unit.moduleActive THEN
       #instEventSum_Status_EM00(In_EventStatus := "EM00".Status,   // "CPG_EventSummation"
                               Sts_EventSummation := "Status".Summation,
                               Sts_NumEvents => #instEventSum_Status_EM00.Sts_NumEvents,
                               Sts_CurrentActiveEvent => #instEventSum_Status_EM00.Sts_CurrentActiveEvent,
                               Sts_Error => #instEventSum_Status_EM00.Sts_Error,
                               Sts_ErrorCode => #instEventSum_Status_EM00.Sts_ErrorCode);
   END_IF;
END_REGION

REGION Network 24: Status Event Summary Logic - Equipment Module #01
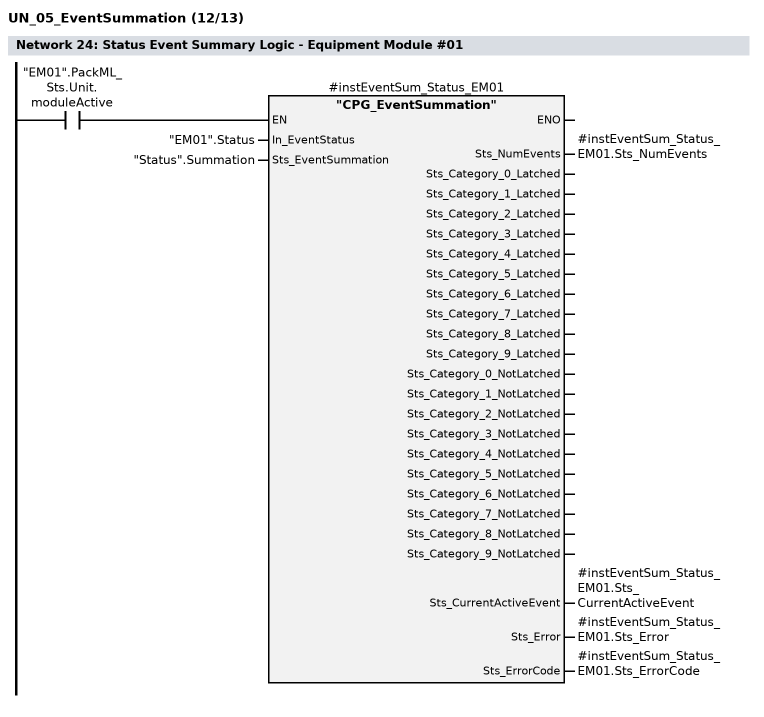
   RUNG wire#powerrail
      Contact( "EM01".PackML_Sts.Unit.moduleActive )
      #instEventSum_Status_EM01(In_EventStatus := "EM01".Status, Sts_EventSummation := "Status".Summation, Sts_NumEvents => #instEventSum_Status_EM01.Sts_NumEvents, Sts_Category_0_Latched =>, Sts_Category_1_Latched =>, Sts_Category_2_Latched =>, Sts_Category_3_Latched =>, Sts_Category_4_Latched =>, Sts_Category_5_Latched =>, Sts_Category_6_Latched =>, Sts_Category_7_Latched =>, Sts_Category_8_Latched =>, Sts_Category_9_Latched =>, Sts_Category_0_NotLatched =>, Sts_Category_1_NotLatched =>, Sts_Category_2_NotLatched =>, Sts_Category_3_NotLatched =>, Sts_Category_4_NotLatched =>, Sts_Category_5_NotLatched =>, Sts_Category_6_NotLatched =>, Sts_Category_7_NotLatched =>, Sts_Category_8_NotLatched =>, Sts_Category_9_NotLatched =>, Sts_CurrentActiveEvent => #instEventSum_Status_EM01.Sts_CurrentActiveEvent, Sts_Error => #instEventSum_Status_EM01.Sts_Error, Sts_ErrorCode => #instEventSum_Status_EM01.Sts_ErrorCode)
   END_RUNG
   // the same network as SCL:
   IF "EM01".PackML_Sts.Unit.moduleActive THEN
       #instEventSum_Status_EM01(In_EventStatus := "EM01".Status,   // "CPG_EventSummation"
                               Sts_EventSummation := "Status".Summation,
                               Sts_NumEvents => #instEventSum_Status_EM01.Sts_NumEvents,
                               Sts_CurrentActiveEvent => #instEventSum_Status_EM01.Sts_CurrentActiveEvent,
                               Sts_Error => #instEventSum_Status_EM01.Sts_Error,
                               Sts_ErrorCode => #instEventSum_Status_EM01.Sts_ErrorCode);
   END_IF;
END_REGION

REGION Network 25: Status Event Summary Logic - Equipment Module #02
   // This instance of the Event Sum (or Event Summation) is used to merge the events 
   // from EM01 into the larger Unit or UN evevts list.
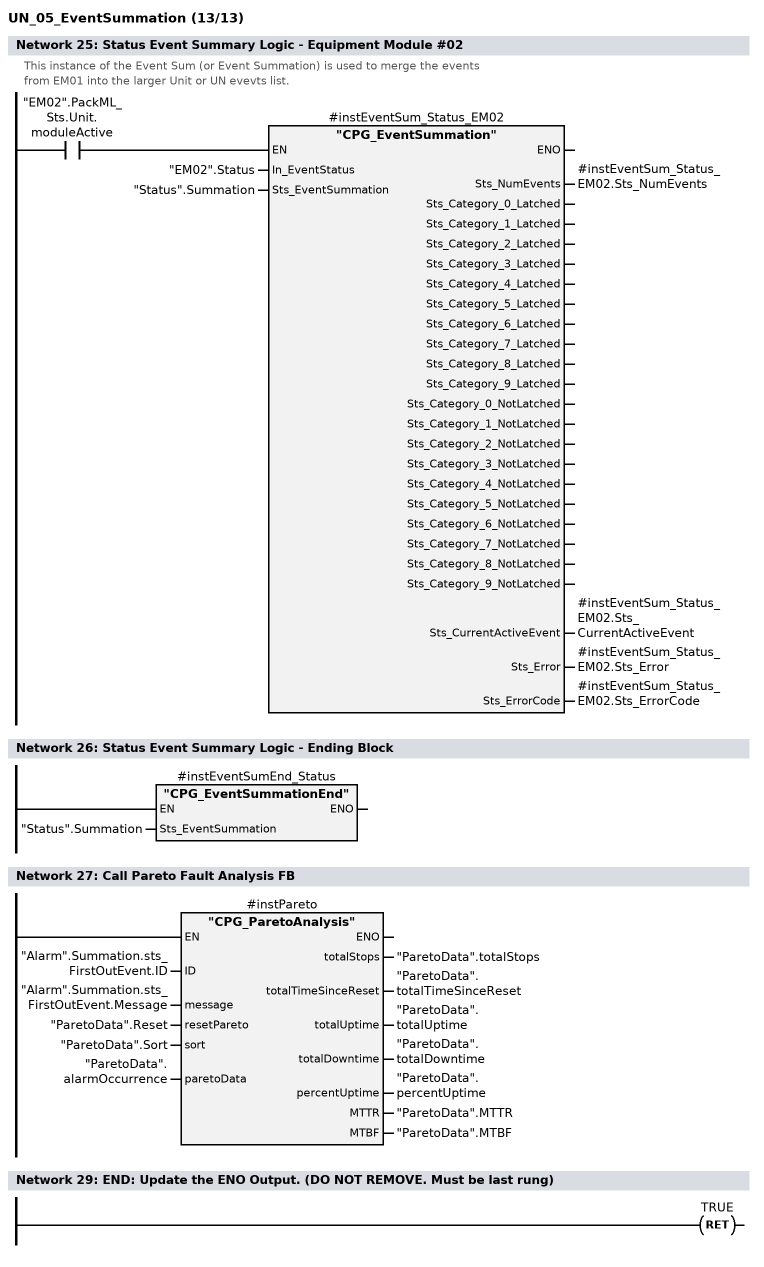
   RUNG wire#powerrail
      Contact( "EM02".PackML_Sts.Unit.moduleActive )
      #instEventSum_Status_EM02(In_EventStatus := "EM02".Status, Sts_EventSummation := "Status".Summation, Sts_NumEvents => #instEventSum_Status_EM02.Sts_NumEvents, Sts_Category_0_Latched =>, Sts_Category_1_Latched =>, Sts_Category_2_Latched =>, Sts_Category_3_Latched =>, Sts_Category_4_Latched =>, Sts_Category_5_Latched =>, Sts_Category_6_Latched =>, Sts_Category_7_Latched =>, Sts_Category_8_Latched =>, Sts_Category_9_Latched =>, Sts_Category_0_NotLatched =>, Sts_Category_1_NotLatched =>, Sts_Category_2_NotLatched =>, Sts_Category_3_NotLatched =>, Sts_Category_4_NotLatched =>, Sts_Category_5_NotLatched =>, Sts_Category_6_NotLatched =>, Sts_Category_7_NotLatched =>, Sts_Category_8_NotLatched =>, Sts_Category_9_NotLatched =>, Sts_CurrentActiveEvent => #instEventSum_Status_EM02.Sts_CurrentActiveEvent, Sts_Error => #instEventSum_Status_EM02.Sts_Error, Sts_ErrorCode => #instEventSum_Status_EM02.Sts_ErrorCode)
   END_RUNG
   // the same network as SCL:
   IF "EM02".PackML_Sts.Unit.moduleActive THEN
       #instEventSum_Status_EM02(In_EventStatus := "EM02".Status,   // "CPG_EventSummation"
                               Sts_EventSummation := "Status".Summation,
                               Sts_NumEvents => #instEventSum_Status_EM02.Sts_NumEvents,
                               Sts_CurrentActiveEvent => #instEventSum_Status_EM02.Sts_CurrentActiveEvent,
                               Sts_Error => #instEventSum_Status_EM02.Sts_Error,
                               Sts_ErrorCode => #instEventSum_Status_EM02.Sts_ErrorCode);
   END_IF;
END_REGION

REGION Network 26: Status Event Summary Logic - Ending Block
   RUNG wire#powerrail
      #instEventSumEnd_Status(Sts_EventSummation := "Status".Summation)
   END_RUNG
   // the same network as SCL:
   #instEventSumEnd_Status(Sts_EventSummation := "Status".Summation);   // "CPG_EventSummationEnd"
END_REGION

REGION Network 27: Call Pareto Fault Analysis FB
   RUNG wire#powerrail
      #instPareto(ID := "Alarm".Summation.sts_FirstOutEvent.ID, message := "Alarm".Summation.sts_FirstOutEvent.Message, resetPareto := "ParetoData".Reset, sort := "ParetoData".Sort, paretoData := "ParetoData".alarmOccurrence, totalStops => "ParetoData".totalStops, totalTimeSinceReset => "ParetoData".totalTimeSinceReset, totalUptime => "ParetoData".totalUptime, totalDowntime => "ParetoData".totalDowntime, percentUptime => "ParetoData".percentUptime, MTTR => "ParetoData".MTTR, MTBF => "ParetoData".MTBF)
   END_RUNG
   // the same network as SCL:
   #instPareto(ID := "Alarm".Summation.sts_FirstOutEvent.ID,   // "CPG_ParetoAnalysis"
               message := "Alarm".Summation.sts_FirstOutEvent.Message,
               resetPareto := "ParetoData".Reset,
               sort := "ParetoData".Sort,
               paretoData := "ParetoData".alarmOccurrence,
               totalStops => "ParetoData".totalStops,
               totalTimeSinceReset => "ParetoData".totalTimeSinceReset,
               totalUptime => "ParetoData".totalUptime,
               totalDowntime => "ParetoData".totalDowntime,
               percentUptime => "ParetoData".percentUptime,
               MTTR => "ParetoData".MTTR,
               MTBF => "ParetoData".MTBF);
END_REGION

REGION Network 28: HMI Warning scroll banner logic
END_REGION

REGION Network 29: END: Update the ENO Output. (DO NOT REMOVE. Must be last rung)
   RUNG wire#powerrail
      ReturnCoil( TRUE )
   END_RUNG
   // the same network as SCL:
   ENO := TRUE;
   RETURN;
END_REGION
END_FUNCTION_BLOCK
